Fanuc KAREL source: kt00913.compact.KL

PROGRAM KT00913
%STACKSIZE=65535
%PRIORITY=65535
%NOLOCKGROUP
VAR
S1 : STRING[80]
S2 : STRING[80]
OUT : INTEGER
BEGIN
S1='A'
S2='B'
S1='A'
S2='B'
OUT=STR_LEN(S1)
END KT00913
